(* IEC 61131-3 sources: RingBufLib/RingBufLib/V0.01.0, 5 files *)

(* ---- RingBuffer.typ ---- *)
(********************************************************************
 * COPYRIGHT -- Automation Resources Group
 ********************************************************************
 * Library: RingBufLib
 * File: RingBuffer.typ
 * Author: David Blackburn
 * Created: November 04, 2011
 ********************************************************************
 * Data types of library RingBufLib
 ********************************************************************)

TYPE
	RingBuffer_Internal_typ : 	STRUCT
		pStart : UDINT;
		BufferLength : UDINT;
		iWrite : UDINT;
		iOldestEntry : UDINT;
		iMax : UDINT;
	END_STRUCT;
	RingBuffer_OUT_STAT_typ : 	STRUCT
		Initialized : BOOL;
		NumEntries : UDINT;
	END_STRUCT;
	RingBuffer_OUT_typ : 	STRUCT
		STAT : RingBuffer_OUT_STAT_typ;
	END_STRUCT;
	RingBuffer_IN_CFG_typ : 	STRUCT
		EntrySize : UDINT;
		MaxEntries : UDINT;
	END_STRUCT;
	RingBuffer_IN_typ : 	STRUCT
		CFG : RingBuffer_IN_CFG_typ;
	END_STRUCT;
	RingBuffer_typ : 	STRUCT
		IN : RingBuffer_IN_typ;
		OUT : RingBuffer_OUT_typ;
		Internal : RingBuffer_Internal_typ;
	END_STRUCT;
END_TYPE

(* ---- RingBufLib.typ ---- *)
(********************************************************************
 * COPYRIGHT -- Automation Resources Group
 ********************************************************************
 * Library: RingBufLib
 * File: RingBufLib.typ
 * Author: David Blackburn
 * Created: November 04, 2011
 ********************************************************************
 * Data types of library RingBufLib
 ********************************************************************)

TYPE

END_TYPE

(* ---- RngBuf_Err.typ ---- *)
(********************************************************************
 * COPYRIGHT -- Automation Resources Group
 ********************************************************************
 * Library: RingBufLib
 * File: RngBuf_Err.typ
 * Author: David Blackburn
 * Created: November 04, 2011
 ********************************************************************
 * Data types of library RingBufLib
 ********************************************************************)

TYPE
	RNGBUF_WARN_enum :
		(
		RNGBUF_WARN_MAXDATALENGTH := 500,
		RNGBUF_WARN_
		);
	RNGBUF_ERR_enum :
		(
		RNGBUF_ERROR := 1000,
		RNGBUF_ERR_BADCFG,
		RNGBUF_ERR_MEMALLOC,
		RNGBUF_ERR_INVALIDINPUT,
		RNGBUF_ERR_BUFFNOTINIT,
		RNGBUF_ERR_CORRUPTBUFFER,
		RNGBUF_ERR_
		);
END_TYPE

(* ---- RingBufLib.fun ---- *)
(********************************************************************
 * COPYRIGHT -- Automation Resources Group
 ********************************************************************
 * Library: RingBufLib
 * File: RingBufLib.fun
 * Author: David Blackburn
 * Created: November 04, 2011
 ********************************************************************
 * Functions and function blocks of library RingBufLib
 ********************************************************************)

FUNCTION rngbuf_Init : UINT (*Initialize the ring buffer. MUST BE CALLED IN INIT ROUTINE.*)
	VAR_IN_OUT
		t : RingBuffer_typ; (*RingBuffer object*)
	END_VAR
END_FUNCTION

FUNCTION rngbuf_Reset : UINT (*Reset the ring buffer to the newly initialized state*)
	VAR_IN_OUT
		t : RingBuffer_typ; (*RingBuffer object*)
	END_VAR
END_FUNCTION

FUNCTION rngbuf_Write : UINT (*Add an entry to the ring buffer*)
	VAR_INPUT
		pEntry : UDINT; (*Pointer to the entry to add to the ring buffer*)
		EntrySize : UDINT; (*Size of the entry to add to the ring buffer. Added as check value. Must match RingBuffer.IN.CFG.EntrySize*)
	END_VAR
	VAR_IN_OUT
		t : RingBuffer_typ; (*RingBuffer object*)
	END_VAR
END_FUNCTION

FUNCTION rngbuf_Read : UINT (*Read entries from the ring buffer*)
	VAR_INPUT
		pDest : UDINT; (*Destination address*)
		MaxDataLength : UDINT; (*Maximum amount of data to copy [bytes]*)
		StartingIndex : UDINT; (*Number of entries before most recent to start reading. 0 implies newest entries. 10 implies 10 entries before the newest entry*)
		NumEntries : UDINT; (*Number of entries to copy [entries]. Limited to RingBuffer.OUT.STAT.NumEntries*)
	END_VAR
	VAR_IN_OUT
		t : RingBuffer_typ; (*RingBuffer object*)
	END_VAR
END_FUNCTION

(* ---- RingBufLib.var ---- *)
(********************************************************************
 * COPYRIGHT -- Automation Resources Group
 ********************************************************************
 * Library: RingBufLib
 * File: RingBufLib.var
 * Author: David Blackburn
 * Created: November 04, 2011
 ********************************************************************
 * Constants of library RingBufLib
 ********************************************************************)
VAR CONSTANT
	RNGBUF_NEWEST : UDINT := 0; (*Min UDINT value to read the newest entries in the buffer*)
	RNGBUF_OLDEST : UDINT := 4294967295; (*Max UDINT value to read the oldest entries in the buffer*)
	RNGBUF_ALL : UDINT := 4294967295; (*Max UDINT value to read all entries in the buffer*)
END_VAR
